TYPE ST_BaseLabel :
STRUCT
	arrText		: ARRAY [1..GVL_BaseConstans.LICZBA_DODANYCH_JEZYKOW] OF WSTRING;
	
END_STRUCT
END_TYPE

(* stored: Version 1.1.0.1
   DUT ST_BaseLabel: Id {a8bc978c-f860-0716-3224-49a452076ff3} *)
